FUNCTION TryConvert_DT_TO_DT : BOOL
VAR_INPUT
	in : DT;
	out : REFERENCE TO DT;
END_VAR

out := in;
TryConvert_DT_TO_DT := TRUE;

END_FUNCTION

(* stored: Version 1.1.0.1, ProductVersion 3.1.4024.12
   POU TryConvert_DT_TO_DT: Id {7b5bc23c-fd27-43e8-a67d-27dbe874f19a}, SpecialFunc None *)
